TYPE ST_AWEA_Out :
STRUCT
	DoorOpen			:BIT;
	DoorClose			:BIT;
	Start				:BIT;
	M401_Ack			:BIT;
	M402_Ack			:BIT;
	M403_Ack			:BIT;
END_STRUCT
END_TYPE

(* stored: Version 1.1.0.1, ProductVersion 3.1.4024.11
   DUT ST_AWEA_Out: Id {dbcd3dd9-aa3d-494c-b956-1375b3d535ec} *)
